(* IEC 61131-3 sources: 2026_Projet_YGO_ExcavatriceDragage/ARCHIVES/20260630_025717/CODE, 7 files *)

(* ---- _TYPES.st ---- *)
// ===== E_DegradationLevel =====
// Enum for system degradation levels
// To be created in CODESYS as a separate POU in _TYPES folder

TYPE E_DegradationLevel :
(
    FULL        := 0,    // All systems operational
    LEVEL1      := 1,    // Encoder OK, Joystick OK, brake degraded
    LEVEL2      := 2,    // Joystick OK, encoder down, manual without position feedback
    MAINTENANCE := 3     // Joystick down or CAN bus dead, machine locked
);
END_TYPE

// ===== ST_BusHealth =====
// Unified bus health structure passed via GVL to all functional FBs
// Consolidates CAN and ETHERCAT status per-equipment

TYPE ST_BusHealth :
STRUCT
    CanHealthy          : BOOL;  // CAN bus and joystick both operational
    EthercatHealthy     : BOOL;  // All 3 ETHERCAT slaves operational
    GlobalHealthy       : BOOL;  // CAN AND ETHERCAT both healthy

    JoystickAvailable   : BOOL;  // Joystick online and operational (CAN)
    EncoderM1Available  : BOOL;  // Encoder M1 online and operational (ETHERCAT)
    EncoderM2Available  : BOOL;  // Encoder M2 online and operational (ETHERCAT)
    VariateurAvailable  : BOOL;  // Variateur online and operational (ETHERCAT)
END_STRUCT
END_TYPE

(* ---- FB_BusAggregator.st ---- *)
FUNCTION_BLOCK FB_BusAggregator
VAR_INPUT
    Enable              : BOOL;

    // CAN bus health (from FB_DiagCanOpen)
    CanOnline           : BOOL;
    CanOperational      : BOOL;
    JoystickOnline      : BOOL;
    JoystickOperational : BOOL;

    // ETHERCAT slave health (from 3x FB_DiagEthercat instances)
    Cod1Online          : BOOL;
    Cod1Operational     : BOOL;
    Cod2Online          : BOOL;
    Cod2Operational     : BOOL;
    VariateurOnline     : BOOL;
    VariateurOperational: BOOL;
END_VAR
VAR_OUTPUT
    Ready               : BOOL;

    // Consolidated bus health
    CanHealthy          : BOOL;       // CanOnline AND CanOperational AND JoystickOperational
    EthercatHealthy     : BOOL;       // All 3 slaves operational (Cod1 AND Cod2 AND Variateur)
    GlobalHealthy       : BOOL;       // CanHealthy AND EthercatHealthy

    // Per-equipment availability (used by functional FBs to determine degradation level)
    JoystickAvailable   : BOOL;
    EncoderM1Available  : BOOL;
    EncoderM2Available  : BOOL;
    VariateurAvailable  : BOOL;
END_VAR

// 🛑 GATE
IF NOT Enable THEN
    Ready := FALSE;
    CanHealthy := FALSE;
    EthercatHealthy := FALSE;
    GlobalHealthy := FALSE;
    JoystickAvailable := FALSE;
    EncoderM1Available := FALSE;
    EncoderM2Available := FALSE;
    VariateurAvailable := FALSE;
    RETURN;
END_IF;

Ready := TRUE;

// 🔍 CAN BUS CONSOLIDATION
CanHealthy := CanOperational AND JoystickOperational;
JoystickAvailable := JoystickOnline AND JoystickOperational;

// 🔍 ETHERCAT CONSOLIDATION
EthercatHealthy :=
    (Cod1Online AND Cod1Operational) AND
    (Cod2Online AND Cod2Operational) AND
    (VariateurOnline AND VariateurOperational);

// Per-equipment availability (can be individually down)
EncoderM1Available := Cod1Online AND Cod1Operational;
EncoderM2Available := Cod2Online AND Cod2Operational;
VariateurAvailable := VariateurOnline AND VariateurOperational;

// 🧾 GLOBAL HEALTH
GlobalHealthy := CanHealthy AND EthercatHealthy;

END_FUNCTION_BLOCK

(* ---- FB_DiagCanOpen.st ---- *)
FUNCTION_BLOCK FB_DiagCanOpen
VAR_INPUT
    Enable              : BOOL;       // Activate monitoring
    Reset               : BOOL;       // Fault acknowledgement (rising edge)
    BusState            : BUS_STATE;  // CAN bus state enum
    BusDiagAvailable    : BOOL;       // Diagnosis info available
    DeviceState         : DEVICE_STATE; // Joystick CANopen node state
    DevDiagAvailable    : BOOL;       // Device diagnosis available
END_VAR
VAR_OUTPUT
    Ready               : BOOL;       // Block operational
    Error               : BOOL;       // Mirror of (ErrorId <> 0)
    ErrorId             : WORD;       // Bitfield: bit0=bus down, bit1=device not found, bit2=device not operational
    BusOnline           : BOOL;       // Bus physically responds
    BusOperational      : BOOL;       // Bus in RUN state
    JoystickOnline      : BOOL;       // Device present on bus
    JoystickOperational : BOOL;       // Device in NMT Operational state
    CanHealthy          : BOOL;       // BusOperational AND JoystickOperational
END_VAR
VAR
    ResetEdge           : R_TRIG;
END_VAR

// 🛑 1. GATE DE SÉCURITÉ
IF NOT Enable THEN
    Ready := FALSE;
    BusOnline := FALSE;
    BusOperational := FALSE;
    JoystickOnline := FALSE;
    JoystickOperational := FALSE;
    CanHealthy := FALSE;
    Error := FALSE;
    ErrorId := 16#0000;
    RETURN;
END_IF;

Ready := TRUE;

// 🔑 2. RESET DÉFAUT (front obligatoire)
ResetEdge(CLK := Reset);
IF ResetEdge.Q THEN
    IF (BusOperational AND JoystickOperational) THEN
        ErrorId := 16#0000;
    END_IF;
END_IF;

// 🔍 3. DIAGNOSTIC BUS CAN
// BusState available → check bus health
BusOnline := (BusState <> BUS_STATE.IDLE); // Bus has activity
BusOperational := (BusState = BUS_STATE.RUNNING); // Bus in RUN mode

IF NOT BusOperational THEN
    ErrorId.0 := TRUE; // bit0: bus down
ELSE
    ErrorId.0 := FALSE;
END_IF;

// 🔍 4. DIAGNOSTIC JOYSTICK NODE
// DeviceState check
JoystickOnline := (DeviceState <> DEVICE_STATE.NOT_FOUND);

IF NOT JoystickOnline THEN
    ErrorId.1 := TRUE; // bit1: device not found
ELSE
    ErrorId.1 := FALSE;
END_IF;

// Device operational state (NMT Operational in CANopen)
JoystickOperational := (DeviceState = DEVICE_STATE.RUNNING);

IF NOT JoystickOperational AND JoystickOnline THEN
    ErrorId.2 := TRUE; // bit2: device not operational
ELSE
    IF JoystickOnline THEN
        ErrorId.2 := FALSE;
    END_IF;
END_IF;

// 🧾 5. CONSOLIDATED OUTPUT
CanHealthy := BusOperational AND JoystickOperational;
Error := (ErrorId <> 16#0000);

END_FUNCTION_BLOCK

(* ---- FB_DiagEthercat_IMPROVED.st ---- *)
FUNCTION_BLOCK FB_DiagEthercat
VAR_INPUT
    Enable          : BOOL;       // Activate monitoring
    Reset           : BOOL;       // Fault acknowledgement (rising edge)
    WcState         : BOOL;       // Working Counter (FALSE = valid frame / online)
    SlaveState      : WORD;       // Internal slave state (8 = OP / Operational)
END_VAR
VAR_OUTPUT
    Ready           : BOOL;       // Block operational
    Online          : BOOL;       // Slave present and responding
    Operational     : BOOL;       // Slave in OP mode (valid data)
    Error           : BOOL;       // Fault active
    ErrorId         : WORD;       // Error code (bit0=offline, bit1=not operational)
    StateAtError    : WORD;       // Snapshot of SlaveState at fault instant (frozen until ack)
END_VAR
VAR
    ResetEdge       : R_TRIG;
    LastSlaveState  : WORD;       // Capture state on fault for StateAtError
END_VAR

// 🛑 1. GATE DE SÉCURITÉ
IF NOT Enable THEN
    Ready := FALSE;
    Online := FALSE;
    Operational := FALSE;
    Error := FALSE;
    ErrorId := 16#0000;
    RETURN;
END_IF;

Ready := TRUE;

// 🔑 2. RESET DÉFAUT (front obligatoire)
ResetEdge(CLK := Reset);

IF ResetEdge.Q THEN
    // Only clear error if cause has disappeared
    IF Online AND Operational THEN
        Error := FALSE;
        ErrorId := 16#0000;
        StateAtError := 0;  // Clear snapshot on successful ack
    END_IF;
END_IF;

// 🔍 3. DIAGNOSTIC ETHERCAT
// WcState à FALSE signifie que le maître communique physiquement avec le nœud
Online := NOT WcState;

// L'état 8 en EtherCAT correspond à l'état "Operational" (échanges cycliques actifs)
Operational := Online AND (SlaveState = 8);

// ⚠️ 4. GESTION DES ERREURS avec snapshot StateAtError
IF NOT Online THEN
    IF NOT Error THEN
        // Transition to error: capture state
        LastSlaveState := SlaveState;
        StateAtError := SlaveState;
    END_IF;
    Error := TRUE;
    ErrorId.0 := TRUE;   // bit0: offline
    ErrorId.1 := FALSE;
ELSIF NOT Operational THEN
    IF NOT Error THEN
        // Transition to error: capture state
        LastSlaveState := SlaveState;
        StateAtError := SlaveState;
    END_IF;
    Error := TRUE;
    ErrorId.0 := FALSE;
    ErrorId.1 := TRUE;   // bit1: not operational
ELSE
    // No error condition
    ErrorId := 16#0000;
END_IF;

END_FUNCTION_BLOCK

(* ---- FB_Encoder_Abs_REFACTORED.st ---- *)
// FB_Encoder_Abs — Refactored version
// Conformance with AF_Partie3 + EtherCAT bus gate + ErrorId bitfield
// Replace the original FB_Encoder_Abs content with this code

FUNCTION_BLOCK FB_Encoder_Abs
VAR_INPUT
    Enable              : BOOL;   // Active la logique
    Reset               : BOOL;   // Acquittement défaut (front obligatoire)
    SafeStop            : BOOL;   // Arrêt sûr forcé
    SafetyOk            : BOOL;   // Conditions globales OK
    EthOnline           : BOOL;   // Esclave EtherCAT présent
    EthOperational      : BOOL;   // Esclave EtherCAT opérationnel

    In_Alarms           : UINT;   // %IW2 — hardware alarm word
    In_Warnings         : UINT;   // %IW3
    In_PosValue         : UDINT;  // %ID2 — raw position
    In_SpdValue         : INT;    // %IW6 — raw speed

    HomingTrigger       : BOOL;   // Rising edge trigger for water level homing
    WaterLevelOffset    : REAL;   // Water level offset in metres

    InvertDirection     : BOOL;   // Mechanical direction inversion
    MaxSpeedThreshold   : INT := 5000;

    TeachActive         : BOOL;   // Calibration mode
    TeachStartRaw       : UDINT;  // Teach point A raw position
    TeachEndRaw         : UDINT;  // Teach point B raw position
    TeachRealDistance   : REAL;   // Measured distance A→B in metres
END_VAR
VAR_OUTPUT
    Ready               : BOOL;   // Block operational
    Busy                : BOOL;   // Processing active
    Done                : BOOL;   // Action complete
    Error               : BOOL;   // Mirror of (ErrorId <> 0)
    ErrorId             : WORD;   // Bitfield: bit0=alarm, bit1=overspeed, bit2=offline, bit3=not operational
    State               : WORD;   // Operational phase (0=disabled, 1=ready, 2=processing)
    StateAtError        : WORD;   // Snapshot of SlaveState at error instant

    Out_PresetCmd       : UINT;   // %QW2 — preset command
    Out_PresetValue     : UDINT;  // %QD2 — preset value to write

    ActualPositionM     : REAL;   // Final position in metres
    ActualSpeedFiltered : REAL;   // Filtered speed for monitoring
    EmergencyStop       : BOOL;   // Immediate braking request (overspeed action)
END_VAR
VAR_IN_OUT
    Config_PulsePerMeter : REAL;  // Persistent calibration
END_VAR
VAR
    GetCycleTime        : FB_CycleTime;
    ScaleStage          : FB_Encoder_Scale;
    SafetyStage         : FB_Encoder_Safety;
    ResetEdge           : R_TRIG;

    LocalRawPos         : UDINT;
    LastHomingTrigger   : BOOL;
    LastSlaveState      : WORD;
END_VAR

// 🛑 1. GATE DE SÉCURITÉ (Prioritaire)
IF NOT Enable OR SafeStop OR NOT EthOnline OR NOT EthOperational THEN
    Ready := FALSE;
    Busy := FALSE;
    Done := FALSE;
    State := 0;  // DISABLED
    Out_PresetCmd := 0;
    Out_PresetValue := 0;
    ActualSpeedFiltered := 0.0;
    EmergencyStop := TRUE;  // Fail-safe
    RETURN;
END_IF;

Ready := TRUE;
State := 1;  // READY

// 🔑 2. RESET DÉFAUT (front obligatoire)
ResetEdge(CLK := Reset);

IF ResetEdge.Q THEN
    // Clear error only if all causes have disappeared
    IF EthOnline AND EthOperational AND (In_Alarms = 0) AND (SafetyStage.OverspeedTrip = FALSE) THEN
        ErrorId := 16#0000;
        Error := FALSE;
        StateAtError := 0;
    END_IF;
END_IF;

// 📥 3. ACQUISITION &amp; CYCLE TIME
GetCycleTime();

// Handle direction inversion
IF InvertDirection THEN
    LocalRawPos := 16#FFFFFFFF - In_PosValue;
ELSE
    LocalRawPos := In_PosValue;
END_IF;

// ⚙️ 4. HOMING / PRESET LOGIC (single implementation)
IF HomingTrigger AND NOT LastHomingTrigger THEN
    Out_PresetValue := REAL_TO_UDINT(WaterLevelOffset * Config_PulsePerMeter);
    Out_PresetCmd := 16#0001;
    Busy := TRUE;
ELSE
    Out_PresetCmd := 16#0000;
    Busy := FALSE;
END_IF;
LastHomingTrigger := HomingTrigger;

// 🧾 5. ERROR DETECTION (bitfield)

// bit0 = hardware alarm
IF (In_Alarms &lt;&gt; 0) THEN
    IF NOT Error THEN
        StateAtError := 1;  // Capture error state
    END_IF;
    ErrorId.0 := TRUE;
ELSE
    ErrorId.0 := FALSE;
END_IF;

// PIPELINE SCALING
ScaleStage(
    CurrentRawPos := LocalRawPos,
    OffsetValueB := 0.0,
    EnableTeach := TeachActive,
    StartTeachPos := TeachStartRaw,
    EndTeachPos := TeachEndRaw,
    RealDistMeters := TeachRealDistance,
    PulsePerMeter := Config_PulsePerMeter
);
ActualPositionM := ScaleStage.PositionMeters;

// PIPELINE SAFETY &amp; SPEED
SafetyStage(
    RawSpeed := In_SpdValue,
    MaxSpeedLimit := MaxSpeedThreshold,
    CycleTimeS := GetCycleTime.CycleTimeS
);
ActualSpeedFiltered := SafetyStage.FilteredSpeed;

// bit1 = overspeed
IF SafetyStage.OverspeedTrip THEN
    IF NOT Error THEN
        StateAtError := 2;
    END_IF;
    ErrorId.1 := TRUE;
ELSE
    ErrorId.1 := FALSE;
END_IF;

// bit2 = EtherCAT offline
IF NOT EthOnline THEN
    IF NOT Error THEN
        StateAtError := 3;
    END_IF;
    ErrorId.2 := TRUE;
ELSE
    ErrorId.2 := FALSE;
END_IF;

// bit3 = EtherCAT not operational
IF NOT EthOperational THEN
    IF NOT Error THEN
        StateAtError := 4;
    END_IF;
    ErrorId.3 := TRUE;
ELSE
    ErrorId.3 := FALSE;
END_IF;

// 6. ERROR OUTPUT &amp; EMERGENCY ACTION
Error := (ErrorId &lt;&gt; 16#0000);
EmergencyStop := SafetyStage.OverspeedTrip OR Error;
Done := NOT Error;

END_FUNCTION_BLOCK

(* ---- FB_Safety_REFACTORED.st ---- *)
// FB_Safety — Refactored version
// Granular equipment availability inputs instead of single EthercatOk BOOL
// ErrorId with per-equipment bits

FUNCTION_BLOCK FB_Safety
VAR_INPUT
    Enable              : BOOL;       // Activate monitoring
    Reset               : BOOL;       // Fault acknowledgement
    EStopArmed          : BOOL;       // Emergency stop TOR (TRUE = OK)
    CanOnline           : BOOL;       // CAN bus operational
    CanOperational      : BOOL;       // CAN bus running
    JoystickAvailable   : BOOL;       // Joystick online and operational
    EncoderM1Available  : BOOL;       // Encoder M1 online and operational
    EncoderM2Available  : BOOL;       // Encoder M2 online and operational
    VariateurAvailable  : BOOL;       // Variateur online and operational
END_VAR
VAR_OUTPUT
    Ready               : BOOL;       // Logique de sécurité opérationnelle
    SafeStop            : BOOL;       // Ordre d'arrêt absolu (TRUE = STOP IMMÉDIAT)
    SafetyOk            : BOOL;       // Feu vert global (TRUE = Autorisation de bouger)
    Error               : BOOL;       // Présence anomalie sécurité
    ErrorId             : WORD;       // Bitfield code de cause
END_VAR
VAR
    ResetEdge           : R_TRIG;
END_VAR

// 1. GATE AUTOMATE
IF NOT Enable THEN
    Ready := FALSE;
    SafeStop := TRUE;             // Sécurité par défaut : arrêt forcé
    SafetyOk := FALSE;
    Error := FALSE;
    ErrorId := 16#0000;
    RETURN;
END_IF;

Ready := TRUE;

// 2. RESET DÉFAUTS (front obligatoire)
ResetEdge(CLK := Reset);

IF ResetEdge.Q THEN
    // Clear only if all conditions are met
    IF EStopArmed AND CanOperational AND JoystickAvailable AND
       EncoderM1Available AND EncoderM2Available AND VariateurAvailable THEN
        Error := FALSE;
        ErrorId := 16#0000;
    END_IF;
END_IF;

// 3. LOGIQUE FAIL-SAFE (Perte de signal = Danger)
// bit0 = Emergency stop activated
IF NOT EStopArmed THEN
    ErrorId.0 := TRUE;
ELSE
    ErrorId.0 := FALSE;
END_IF;

// bit1 = CAN bus down
IF NOT CanOperational THEN
    ErrorId.1 := TRUE;
ELSE
    ErrorId.1 := FALSE;
END_IF;

// bit2 = Joystick not available
IF NOT JoystickAvailable THEN
    ErrorId.2 := TRUE;
ELSE
    ErrorId.2 := FALSE;
END_IF;

// bit3 = Encoder M1 down
IF NOT EncoderM1Available THEN
    ErrorId.3 := TRUE;
ELSE
    ErrorId.3 := FALSE;
END_IF;

// bit4 = Encoder M2 down
IF NOT EncoderM2Available THEN
    ErrorId.4 := TRUE;
ELSE
    ErrorId.4 := FALSE;
END_IF;

// bit5 = Variateur down
IF NOT VariateurAvailable THEN
    ErrorId.5 := TRUE;
ELSE
    ErrorId.5 := FALSE;
END_IF;

// 4. ARBITRAGE DES SORTIES TRANSVERSES
Error := (ErrorId &lt;&gt; 16#0000);

// SafeStop est l'actionneur logiciel (TRUE = On coupe tout)
SafeStop := Error;

// SafetyOk est le feu vert (TRUE = Tout est sain)
SafetyOk := NOT Error;

END_FUNCTION_BLOCK

(* ---- PRG_BusMonitor.st ---- *)
// PROGRAM PRG_BusMonitor
// System program: centralizes bus diagnostics and health monitoring
// Calls: FB_DiagCanOpen + 3x FB_DiagEthercat + FB_BusAggregator
// Updates: GVL_BusHealth with consolidated health status
// Task: MainTask (20ms) or CanTask (10ms) depending on bus polling speed

PROGRAM PRG_BusMonitor
VAR
    // ===== DIAGNOSTIC INSTANCES =====
    DiagCanOpen        : FB_DiagCanOpen;
    DiagEthEncoderM1   : FB_DiagEthercat;
    DiagEthEncoderM2   : FB_DiagEthercat;
    DiagEthVariateur   : FB_DiagEthercat;

    // ===== AGGREGATION INSTANCE =====
    BusAggregator      : FB_BusAggregator;

    // ===== ENABLE FLAG =====
    DiagnosticsEnabled : BOOL := TRUE;
END_VAR

// ========================================
// 1. CAN BUS DIAGNOSTIC
// ========================================
DiagCanOpen(
    Enable := DiagnosticsEnabled,
    Reset := GVL_DEBUG.DBG_ResetBusHealth,  // or button from IHM
    BusState := CANopen_Manager.GetBusState(...),  // Provide actual bus state
    BusDiagAvailable := TRUE,                      // Assume available
    DeviceState := JOY1_JOYSTICK_MCB560_CO4201A.GetDeviceState(...),  // Joystick node
    DevDiagAvailable := TRUE
);

// ========================================
// 2. ETHERCAT DIAGNOSTICS (3 slaves)
// ========================================

// Encoder M1 (Treuil M1)
DiagEthEncoderM1(
    Enable := DiagnosticsEnabled,
    Reset := GVL_DEBUG.DBG_ResetBusHealth,
    WcState := CoE_Encoder1_WcState,      // EtherCAT Working Counter state
    SlaveState := CoE_Encoder1_State      // Slave operational state
);

// Encoder M2 (Treuil M2)
DiagEthEncoderM2(
    Enable := DiagnosticsEnabled,
    Reset := GVL_DEBUG.DBG_ResetBusHealth,
    WcState := CoE_Encoder2_WcState,
    SlaveState := CoE_Encoder2_State
);

// Variateur (Translation or other ETHERCAT device)
DiagEthVariateur(
    Enable := DiagnosticsEnabled,
    Reset := GVL_DEBUG.DBG_ResetBusHealth,
    WcState := CoE_Variateur_WcState,
    SlaveState := CoE_Variateur_State
);

// ========================================
// 3. BUS AGGREGATION
// ========================================
BusAggregator(
    Enable := DiagnosticsEnabled,

    // CAN inputs from DiagCanOpen
    CanOnline := DiagCanOpen.BusOnline,
    CanOperational := DiagCanOpen.BusOperational,
    JoystickOnline := DiagCanOpen.JoystickOnline,
    JoystickOperational := DiagCanOpen.JoystickOperational,

    // ETHERCAT inputs from 3x DiagEthercat
    Cod1Online := DiagEthEncoderM1.Online,
    Cod1Operational := DiagEthEncoderM1.Operational,
    Cod2Online := DiagEthEncoderM2.Online,
    Cod2Operational := DiagEthEncoderM2.Operational,
    VariateurOnline := DiagEthVariateur.Online,
    VariateurOperational := DiagEthVariateur.Operational
);

// ========================================
// 4. UPDATE GLOBAL HEALTH STRUCTURE (GVL)
// ========================================
GVL_BusHealth.BusHealth.CanHealthy := BusAggregator.CanHealthy;
GVL_BusHealth.BusHealth.EthercatHealthy := BusAggregator.EthercatHealthy;
GVL_BusHealth.BusHealth.GlobalHealthy := BusAggregator.GlobalHealthy;
GVL_BusHealth.BusHealth.JoystickAvailable := BusAggregator.JoystickAvailable;
GVL_BusHealth.BusHealth.EncoderM1Available := BusAggregator.EncoderM1Available;
GVL_BusHealth.BusHealth.EncoderM2Available := BusAggregator.EncoderM2Available;
GVL_BusHealth.BusHealth.VariateurAvailable := BusAggregator.VariateurAvailable;

END_PROGRAM
